FUNCTION_BLOCK FB_SRAlarm EXTENDS FB_AlarmBase
VAR_INPUT
	bSet					: BOOL;
	bReset					: BOOL;
END_VAR
VAR
	fbSetRTrig				: R_TRIG;
	fbSetFTrig				: F_TRIG;
	fbAckRTrig				: R_TRIG;
END_VAR
VAR_TEMP
	bThisAlarmSelected		: BOOL;
	bAck					: BOOL;
END_VAR

fbSetRTrig(CLK := bSet);
fbSetFTrig(CLK := bSet);

fbAckRTrig(CLK := iAlarmContext.Acknowledge);

IF fbSetRTrig.Q THEN
	iAlarmContext.EnableAcknowledge(nAlarmContextId, FALSE);
END_IF

IF fbSetFTrig.Q THEN
	iAlarmContext.EnableAcknowledge(nAlarmContextId, TRUE);
END_IF

bThisAlarmSelected := iAlarmContext.SelectedAlarmContextId <> ALARM_INVALID_CONTEXT_ID AND
	nAlarmContextId <> ALARM_INVALID_CONTEXT_ID AND
	iAlarmContext.SelectedAlarmContextId = nAlarmContextId;
	
bAck := bThisAlarmSelected AND fbAckRTrig.Q;

bActive := (NOT bReset AND NOT bAck AND bActive) OR bSet;

SUPER^();

PROPERTY ArgStackMemoryPointer : POINTER TO BYTE
GET
ArgStackMemoryPointer := 0;
END_GET
END_PROPERTY

PROPERTY ArgStackMemorySize : DINT
GET
ArgStackMemorySize := 0;
END_GET
END_PROPERTY

METHOD PROTECTED  ClearArgStack
VAR_INPUT
END_VAR
// Do nothing
END_METHOD

METHOD PROTECTED CopyArgsToStack
VAR_INPUT
END_VAR
// Do nothing
END_METHOD

END_FUNCTION_BLOCK

(* stored: Version 1.1.0.1, ProductVersion 3.1.4024.15
   POU FB_SRAlarm: Id {45bb9f76-c2ac-4273-b2d4-b673bb9a0f2c}, SpecialFunc None
   Property ArgStackMemoryPointer: Id {061a69c4-944e-4d0a-a770-a48d503e36d6}
   Get Get: Id {76da89dc-b20a-458a-91ff-eb7160c72dc2}
   Property ArgStackMemorySize: Id {ce492647-c1b1-4e4c-8df4-e89f72b98e2f}
   Get Get: Id {6352f1f8-46de-4bd0-87d2-4d81c3ad9a20}
   Method ClearArgStack: Id {c4c5d467-dffb-41bb-be6f-9a38b3bc597d}
   Method CopyArgsToStack: Id {185a466b-e503-4527-9e7c-4eca1b3d7041} *)
